{attribute 'qualified_only'}
VAR_GLOBAL
END_VAR

(* stored: Version 1.1.0.1, ProductVersion 3.1.4022.16
   GVL GVL: Id {2d665628-afb2-4dd7-ac9b-db077f9b2823} *)
